ABB RobotStudio station: Eksamens_20200508-111548.rsstn

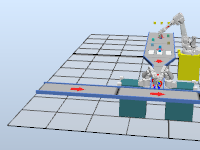
Station Eksamens (saved by RobotStudio 7.0.8746.631)
Controller Virtual_controller, task T_ROB3: task frame (RAPID world) sits at (-5805.06, 703.5, 890) mm, rotated rx 0 ry 0 rz -90 deg in the station
Controller Virtual_controller, task T_ROB2: task frame (RAPID world) sits at (-5805.06, 703.5, 890) mm, rotated rx 0 ry 0 rz -90 deg in the station
Controller Virtual_controller, task T_ROB1: task frame (RAPID world) sits at (-5805.06, 703.5, 890) mm, rotated rx 0 ry 0 rz -90 deg in the station
Controller Virtual_controller
  mechanical unit ROB_1: IRB120_3_58__01_2, 6 joints, base frame (83.5, -144.94, 0) mm
  mechanical unit ROB_2: IRB2600_20_165_C_01_2, 6 joints, base frame (1331.39, 3332.7, 0) mm, rotated rx 0 ry 0 rz 180 deg
  mechanical unit ROB_3: IRB120_3_58__01_3, 6 joints, base frame (643.5, -144.94, 0) mm, rotated rx 0 ry 0 rz 180 deg
Layout (positions relative to the parent item):
  - Sorter_kasser [graphiccomponentgroup]
    - Assemblies [graphiccomponentgroup]
      - Section1 [graphiccomponentgroup]
        - ABB_IRC5_ctrl [graphiccomponentgroup]
          - ABB_IRC5_ctrl_1 [graphiccomponentgroup]
            - Mesh0 [part]
        - Conveyor__Straight_ [graphiccomponentgroup]
          - CONVEYOR1 [graphiccomponentgroup]
            - Mesh1 [part]
            - Mesh2 [part]
            - Mesh3 [part]
          - CONVEYOR2 [graphiccomponentgroup]
            - Mesh4 [part]
            - Mesh5 [part]
            - Mesh6 [part]
          - CONVEYOR3 [graphiccomponentgroup]
            - Mesh7 [part]
            - Mesh8 [part]
            - Mesh9 [part]
          - CONVEYOR4 [graphiccomponentgroup]
            - Mesh10 [part]
            - Mesh11 [part]
            - Mesh12 [part]
          - CONVEYOR5 [graphiccomponentgroup]
            - Mesh13 [part]
            - Mesh14 [part]
            - Mesh15 [part]
          - CONVEYOR6 [graphiccomponentgroup]
            - Mesh16 [part]
            - Mesh17 [part]
            - Mesh18 [part]
          - CONVEYOR7 [graphiccomponentgroup]
            - Mesh19 [part]
            - Mesh20 [part]
            - Mesh21 [part]
        - Cube [graphiccomponentgroup]
          - Cube1 [graphiccomponentgroup]
            - Mesh22 [part]
            - Mesh23 [part]
            - Mesh24 [part]
            - Mesh25 [part]
            - Mesh26 [part]
          - Cube2 [graphiccomponentgroup]
            - Mesh27 [part]
            - Mesh28 [part]
            - Mesh29 [part]
            - Mesh30 [part]
            - Mesh31 [part]
          - Cube3 [graphiccomponentgroup]
            - Mesh32 [part]
            - Mesh33 [part]
            - Mesh34 [part]
            - Mesh35 [part]
            - Mesh36 [part]
        - Eater [graphiccomponentgroup]
          - EATER1 [graphiccomponentgroup]
            - Mesh37 [part]
        - Display [graphiccomponentgroup]
          - EaterSmall [graphiccomponentgroup]
            - Mesh38 [part]
            - Mesh39 [part]
            - Mesh40 [part]
            - Mesh41 [part]
            - Mesh42 [part]
            - Mesh43 [part]
            - Mesh44 [part]
            - Mesh45 [part]
            - Mesh46 [part]
            - Mesh47 [part]
            - Mesh48 [part]
        - Feeder [graphiccomponentgroup]
          - FEEDER1 [graphiccomponentgroup]
            - Mesh49 [part]
            - Mesh50 [part]
          - FEEDER2 [graphiccomponentgroup]
            - Mesh51 [part]
            - Mesh52 [part]
          - FEEDER3 [graphiccomponentgroup]
            - Mesh53 [part]
            - Mesh54 [part]
        - Scale [graphiccomponentgroup]
          - Scale_Weight [graphiccomponentgroup]
            - Mesh55 [part]
            - Mesh56 [part]
            - Mesh57 [part]
            - Mesh58 [part]
          - Scale_Weight1 [graphiccomponentgroup]
            - Mesh59 [part]
            - Mesh60 [part]
            - Mesh61 [part]
            - Mesh62 [part]
          - Scale_Weight2 [graphiccomponentgroup]
            - Mesh63 [part]
            - Mesh64 [part]
            - Mesh65 [part]
            - Mesh66 [part]
        - Text [graphiccomponentgroup]
          - Text1 [graphiccomponentgroup]
            - Mesh67 [part]
    - Motors [graphiccomponentgroup]
      - Surface [graphiccomponentgroup]
        - MOTOR1 [graphiccomponentgroup]
          - Mesh75 [part]
          - Mesh76 [part]
          - Mesh77 [part]
          - Mesh78 [part]
        - MOTOR6 [graphiccomponentgroup]
          - Mesh79 [part]
        - MOTOR8 [graphiccomponentgroup]
          - Mesh80 [part]
        - MOTOR9 [graphiccomponentgroup]
          - Mesh81 [part]
    - Loads [graphiccomponentgroup]
      - Mesh68 [part]
      - Mesh69 [part]
      - Mesh70 [part]
      - Mesh71 [part]
      - Mesh72 [part]
      - Mesh73 [part]
      - Mesh74 [part]
  - IRB120_3_58__01_2 [mechanism, from Robots\IRB120_3_58_G_01.rslib] at (-5950, 620, 890) mm, rotated rx 0 ry 0 rz -90 deg; joint values [-1.1313, 0.948, -0.5808, 0, 1.2036, -1.1313] (rad or m)
  - IRB2600_20_165_C_01_2 [mechanism, from Robots\IRB2600_20_165_C_01.rslib] at (-2472.36, -627.89, 890) mm, rotated rx 0 ry 0 rz 90 deg; joint values [0, 0.2407, 0.4991, 6.2832, 0.831, 0] (rad or m)
  - IRB120_3_58__01_3 [mechanism, from Robots\IRB120_3_58_G_01.rslib] at (-5950, 60, 890) mm, rotated rx 0 ry 0 rz 90 deg; joint values [1.0141, 0.7706, 0.0939, 0, 0.7063, 1.0141] (rad or m)
  - GripperStackerRight [mechanism] at (-6426.3, 396.09, 1222.41) mm, rotated rx -180 ry 0 rz 90 deg
      TCP GripperStackerRight at (0, 0, 30) mm
      links: SimpleGripper
  - GripperStackerLeft [mechanism] at (-6321.3, 291.09, 1117.41) mm, rotated rx 180 ry 0 rz -90 deg
      TCP GripperStackerLeft at (0, 0, 30) mm
      links: SimpleGripper
  - GripperSorter [mechanism] at (-2472.36, 353.71, 1478.82) mm, rotated rx 180 ry 0 rz -90 deg
      TCP GripperSorter at (0, 0, 30) mm
      links: SimpleGripper_2
Attachment: GripperStackerRight is attached to IRB120_3_58__01_2 / Link6
Attachment: GripperStackerLeft is attached to IRB120_3_58__01_3 / Link6
Attachment: GripperSorter is attached to IRB2600_20_165_C_01_2 / Link6
Targets, tools, work objects and paths stored in the station, written as RAPID:
! task T_ROB1
MODULE Module1
  CONST robtarget Right22:=[[307.41371826,-621.243232589,302.406306656],[-0.000000055,-0.000000188,1,-0.000000134],[0,-1,0,0],[9E+09,9E+09,9E+09,9E+09,9E+09,9E+09]];
  CONST robtarget Right11:=[[307.41366723,-516.243260729,197.406294596],[-0.000000055,-0.000000188,1,0.000000134],[0,-1,0,0],[9E+09,9E+09,9E+09,9E+09,9E+09,9E+09]];
  CONST robtarget Right12:=[[307.41370671,-621.243260729,197.406322736],[-0.000000055,-0.000000188,1,0.000000134],[0,-1,0,0],[9E+09,9E+09,9E+09,9E+09,9E+09,9E+09]];
  CONST robtarget Right21:=[[307.41367878,-516.243232589,302.406334796],[-0.000000055,-0.000000188,1,-0.000000134],[0,-1,0,0],[9E+09,9E+09,9E+09,9E+09,9E+09,9E+09]];
ENDMODULE

! task T_ROB1
MODULE CalibData
  PERS tooldata GripperStackerRight:=[TRUE,[[0,0,30],[1,0,0,0]],[1,[0,0,1],[1,0,0,0],0,0,0]];
ENDMODULE

! task T_ROB2
MODULE CalibData
  PERS tooldata GripperSorter:=[TRUE,[[0,0,30],[1,0,0,0]],[1,[0,0,1],[1,0,0,0],0,0,0]];
ENDMODULE

! task T_ROB3
MODULE Module1
  CONST robtarget Left12:=[[412.41370671,-621.243221249,197.406311186],[0.000000134,1,0.000000188,-0.000000055],[0,-1,0,0],[9E+09,9E+09,9E+09,9E+09,9E+09,9E+09]];
  CONST robtarget Left11:=[[412.41366723,-516.243221249,197.406283046],[0.000000134,1,0.000000188,-0.000000055],[0,-1,0,0],[9E+09,9E+09,9E+09,9E+09,9E+09,9E+09]];
  CONST robtarget Left22:=[[412.41371826,-621.243193109,302.406295106],[-0.000000134,1,0.000000188,-0.000000055],[0,-1,0,0],[9E+09,9E+09,9E+09,9E+09,9E+09,9E+09]];
  CONST robtarget Left21:=[[412.41367878,-516.243193109,302.406323246],[-0.000000134,1,0.000000188,-0.000000055],[0,-1,0,0],[9E+09,9E+09,9E+09,9E+09,9E+09,9E+09]];
ENDMODULE

! task T_ROB3
MODULE CalibData
  PERS tooldata GripperStackerLeft:=[TRUE,[[0,0,30],[1,0,0,0]],[1,[0,0,1],[1,0,0,0],0,0,0]];
ENDMODULE

